# EPICS substitutions: EUROTHRM/EUROTHRM-IOC-01App/Db/devEurothrmA010.substitutions
# Note: this file is generated by generate_substitutions.py
file devEurothrm.template {
pattern { P, GAD, LAD, MODBUS_PV, MODBUS_SP, MODBUS_P, MODBUS_I, MODBUS_D, MODBUS_HS, MODBUS_LS, MODBUS_AT, MODBUS_HO, MODBUS_OP }
{ "\$(P)", "1", "0", "9217", "9218", "9222", "9224", "9225", "9327", "9328", "9486", "9246", "9219" }
}
